TYPE ST_CYLINDER_IN :
STRUCT
	bEnable				: BOOL;
	bRelExtend			: BOOL;
	bRelRetract			: BOOL;
END_STRUCT
END_TYPE

(* stored: Version 1.1.0.1
   DUT ST_CYLINDER_IN: Id {5f59030a-1b46-4c2d-bcb7-c69fdf9227ec} *)
